(* IEC 61131-3 sources: AXOpen/src/components.abb.robotics/app/src/IO/PLC_LINE, 7 files *)

(* ---- HwIdentifiers.st ---- *)
TYPE
    HwIdentifiers : WORD
    (
        OmniCore_HwID :=	WORD#259,
        OmniCore_DI_64_bytes_DI_64_bytes_HwID :=	WORD#263,
        OmniCore_DO_64_bytes_DO_64_bytes_HwID :=	WORD#262,
        OmniCore_OmniCore_HwID :=	WORD#261,
        OmniCore_OmniCore_OmniCore_Standard_PROFINET_Device_HwID :=	WORD#264,
        OmniCore_OmniCore_profinet_HwID :=	WORD#257,
        OmniCore_OmniCore_profinet_Network_Port_1_HwID :=	WORD#258,
        OmniCore_Rack_HwID :=	WORD#260,
        PROFINET_IO_System_HwID :=	WORD#256,
        RobotBasicIO_HwID :=	WORD#267,
        RobotBasicIO_DI_64_bytes_DI_64_bytes_HwID :=	WORD#271,
        RobotBasicIO_DO_64_bytes_DO_64_bytes_HwID :=	WORD#270,
        RobotBasicIO_Rack_HwID :=	WORD#268,
        RobotBasicIO_RobotBasicIO_HwID :=	WORD#269,
        RobotBasicIO_RobotBasicIO_Robot_Basic_Device_HwID :=	WORD#272,
        RobotBasicIO_RobotBasicIO_profinet_HwID :=	WORD#265,
        RobotBasicIO_RobotBasicIO_profinet_Network_Port_HwID :=	WORD#266,
        plc_line_HwID :=	WORD#32,
        plc_line_Rail_0_HwID :=	WORD#273,
        plc_line_plc_line_HwID :=	WORD#48,
        plc_line_plc_line_CPU_display_1_HwID :=	WORD#54,
        plc_line_plc_line_Card_reader_writer_1_HwID :=	WORD#51,
        plc_line_plc_line_DP_interface_1_HwID :=	WORD#60,
        plc_line_plc_line_OPC_UA_1_HwID :=	WORD#117,
        plc_line_plc_line_PROFINET_interface_X1_HwID :=	WORD#64,
        plc_line_plc_line_PROFINET_interface_X1_Port_1_HwID :=	WORD#65,
        plc_line_plc_line_PROFINET_interface_X1_Port_2_HwID :=	WORD#66,
        plc_line_plc_line_PROFINET_interface_X2_HwID :=	WORD#72,
        plc_line_plc_line_PROFINET_interface_X2_Port_3_HwID :=	WORD#73,
        plc_line_plc_line_Virtual_communication_interface_HwID :=	WORD#135,
        plc_line_plc_line_plc_line_HwID :=	WORD#50,

        NONE := WORD#0
    );
END_TYPE

(* ---- HwInputs.st ---- *)
TYPE
	HwInputs : STRUCT
		RobotBasicIO_DI_64_bytes_1 AT %B0 : ARRAY[0..63] OF BYTE;
		OmniCore_DI_64_bytes_1 AT %B64 : ARRAY[0..63] OF BYTE;
	END_STRUCT;
END_TYPE

(* ---- HwOutputs.st ---- *)
TYPE
	HwOutputs : STRUCT
		RobotBasicIO_DO_64_bytes_1 AT %B0 : ARRAY[0..63] OF BYTE;
		OmniCore_DO_64_bytes_1 AT %B64 : ARRAY[0..63] OF BYTE;
	END_STRUCT;
END_TYPE

(* ---- PlcInputs.st ---- *)
TYPE
	PlcInputs : STRUCT
		RobotBasicIO_DI_64_bytes_1 : ARRAY[0..63] OF BYTE;
		OmniCore_DI_64_bytes_1 : ARRAY[0..63] OF BYTE;
	END_STRUCT;
END_TYPE

(* ---- PlcOutputs.st ---- *)
TYPE
	PlcOutputs : STRUCT
		RobotBasicIO_DO_64_bytes_1 : ARRAY[0..63] OF BYTE;
		OmniCore_DO_64_bytes_1 : ARRAY[0..63] OF BYTE;
	END_STRUCT;
END_TYPE

(* ---- CopyInputs.st ---- *)
FUNCTION CopyInputs
	VAR_EXTERNAL
		HwInputs : HwInputs;
		PlcInputs : PlcInputs;
	END_VAR
	PlcInputs.RobotBasicIO_DI_64_bytes_1[0] := HwInputs.RobotBasicIO_DI_64_bytes_1[0];
	PlcInputs.RobotBasicIO_DI_64_bytes_1[1] := HwInputs.RobotBasicIO_DI_64_bytes_1[1];
	PlcInputs.RobotBasicIO_DI_64_bytes_1[2] := HwInputs.RobotBasicIO_DI_64_bytes_1[2];
	PlcInputs.RobotBasicIO_DI_64_bytes_1[3] := HwInputs.RobotBasicIO_DI_64_bytes_1[3];
	PlcInputs.RobotBasicIO_DI_64_bytes_1[4] := HwInputs.RobotBasicIO_DI_64_bytes_1[4];
	PlcInputs.RobotBasicIO_DI_64_bytes_1[5] := HwInputs.RobotBasicIO_DI_64_bytes_1[5];
	PlcInputs.RobotBasicIO_DI_64_bytes_1[6] := HwInputs.RobotBasicIO_DI_64_bytes_1[6];
	PlcInputs.RobotBasicIO_DI_64_bytes_1[7] := HwInputs.RobotBasicIO_DI_64_bytes_1[7];
	PlcInputs.RobotBasicIO_DI_64_bytes_1[8] := HwInputs.RobotBasicIO_DI_64_bytes_1[8];
	PlcInputs.RobotBasicIO_DI_64_bytes_1[9] := HwInputs.RobotBasicIO_DI_64_bytes_1[9];
	PlcInputs.RobotBasicIO_DI_64_bytes_1[10] := HwInputs.RobotBasicIO_DI_64_bytes_1[10];
	PlcInputs.RobotBasicIO_DI_64_bytes_1[11] := HwInputs.RobotBasicIO_DI_64_bytes_1[11];
	PlcInputs.RobotBasicIO_DI_64_bytes_1[12] := HwInputs.RobotBasicIO_DI_64_bytes_1[12];
	PlcInputs.RobotBasicIO_DI_64_bytes_1[13] := HwInputs.RobotBasicIO_DI_64_bytes_1[13];
	PlcInputs.RobotBasicIO_DI_64_bytes_1[14] := HwInputs.RobotBasicIO_DI_64_bytes_1[14];
	PlcInputs.RobotBasicIO_DI_64_bytes_1[15] := HwInputs.RobotBasicIO_DI_64_bytes_1[15];
	PlcInputs.RobotBasicIO_DI_64_bytes_1[16] := HwInputs.RobotBasicIO_DI_64_bytes_1[16];
	PlcInputs.RobotBasicIO_DI_64_bytes_1[17] := HwInputs.RobotBasicIO_DI_64_bytes_1[17];
	PlcInputs.RobotBasicIO_DI_64_bytes_1[18] := HwInputs.RobotBasicIO_DI_64_bytes_1[18];
	PlcInputs.RobotBasicIO_DI_64_bytes_1[19] := HwInputs.RobotBasicIO_DI_64_bytes_1[19];
	PlcInputs.RobotBasicIO_DI_64_bytes_1[20] := HwInputs.RobotBasicIO_DI_64_bytes_1[20];
	PlcInputs.RobotBasicIO_DI_64_bytes_1[21] := HwInputs.RobotBasicIO_DI_64_bytes_1[21];
	PlcInputs.RobotBasicIO_DI_64_bytes_1[22] := HwInputs.RobotBasicIO_DI_64_bytes_1[22];
	PlcInputs.RobotBasicIO_DI_64_bytes_1[23] := HwInputs.RobotBasicIO_DI_64_bytes_1[23];
	PlcInputs.RobotBasicIO_DI_64_bytes_1[24] := HwInputs.RobotBasicIO_DI_64_bytes_1[24];
	PlcInputs.RobotBasicIO_DI_64_bytes_1[25] := HwInputs.RobotBasicIO_DI_64_bytes_1[25];
	PlcInputs.RobotBasicIO_DI_64_bytes_1[26] := HwInputs.RobotBasicIO_DI_64_bytes_1[26];
	PlcInputs.RobotBasicIO_DI_64_bytes_1[27] := HwInputs.RobotBasicIO_DI_64_bytes_1[27];
	PlcInputs.RobotBasicIO_DI_64_bytes_1[28] := HwInputs.RobotBasicIO_DI_64_bytes_1[28];
	PlcInputs.RobotBasicIO_DI_64_bytes_1[29] := HwInputs.RobotBasicIO_DI_64_bytes_1[29];
	PlcInputs.RobotBasicIO_DI_64_bytes_1[30] := HwInputs.RobotBasicIO_DI_64_bytes_1[30];
	PlcInputs.RobotBasicIO_DI_64_bytes_1[31] := HwInputs.RobotBasicIO_DI_64_bytes_1[31];
	PlcInputs.RobotBasicIO_DI_64_bytes_1[32] := HwInputs.RobotBasicIO_DI_64_bytes_1[32];
	PlcInputs.RobotBasicIO_DI_64_bytes_1[33] := HwInputs.RobotBasicIO_DI_64_bytes_1[33];
	PlcInputs.RobotBasicIO_DI_64_bytes_1[34] := HwInputs.RobotBasicIO_DI_64_bytes_1[34];
	PlcInputs.RobotBasicIO_DI_64_bytes_1[35] := HwInputs.RobotBasicIO_DI_64_bytes_1[35];
	PlcInputs.RobotBasicIO_DI_64_bytes_1[36] := HwInputs.RobotBasicIO_DI_64_bytes_1[36];
	PlcInputs.RobotBasicIO_DI_64_bytes_1[37] := HwInputs.RobotBasicIO_DI_64_bytes_1[37];
	PlcInputs.RobotBasicIO_DI_64_bytes_1[38] := HwInputs.RobotBasicIO_DI_64_bytes_1[38];
	PlcInputs.RobotBasicIO_DI_64_bytes_1[39] := HwInputs.RobotBasicIO_DI_64_bytes_1[39];
	PlcInputs.RobotBasicIO_DI_64_bytes_1[40] := HwInputs.RobotBasicIO_DI_64_bytes_1[40];
	PlcInputs.RobotBasicIO_DI_64_bytes_1[41] := HwInputs.RobotBasicIO_DI_64_bytes_1[41];
	PlcInputs.RobotBasicIO_DI_64_bytes_1[42] := HwInputs.RobotBasicIO_DI_64_bytes_1[42];
	PlcInputs.RobotBasicIO_DI_64_bytes_1[43] := HwInputs.RobotBasicIO_DI_64_bytes_1[43];
	PlcInputs.RobotBasicIO_DI_64_bytes_1[44] := HwInputs.RobotBasicIO_DI_64_bytes_1[44];
	PlcInputs.RobotBasicIO_DI_64_bytes_1[45] := HwInputs.RobotBasicIO_DI_64_bytes_1[45];
	PlcInputs.RobotBasicIO_DI_64_bytes_1[46] := HwInputs.RobotBasicIO_DI_64_bytes_1[46];
	PlcInputs.RobotBasicIO_DI_64_bytes_1[47] := HwInputs.RobotBasicIO_DI_64_bytes_1[47];
	PlcInputs.RobotBasicIO_DI_64_bytes_1[48] := HwInputs.RobotBasicIO_DI_64_bytes_1[48];
	PlcInputs.RobotBasicIO_DI_64_bytes_1[49] := HwInputs.RobotBasicIO_DI_64_bytes_1[49];
	PlcInputs.RobotBasicIO_DI_64_bytes_1[50] := HwInputs.RobotBasicIO_DI_64_bytes_1[50];
	PlcInputs.RobotBasicIO_DI_64_bytes_1[51] := HwInputs.RobotBasicIO_DI_64_bytes_1[51];
	PlcInputs.RobotBasicIO_DI_64_bytes_1[52] := HwInputs.RobotBasicIO_DI_64_bytes_1[52];
	PlcInputs.RobotBasicIO_DI_64_bytes_1[53] := HwInputs.RobotBasicIO_DI_64_bytes_1[53];
	PlcInputs.RobotBasicIO_DI_64_bytes_1[54] := HwInputs.RobotBasicIO_DI_64_bytes_1[54];
	PlcInputs.RobotBasicIO_DI_64_bytes_1[55] := HwInputs.RobotBasicIO_DI_64_bytes_1[55];
	PlcInputs.RobotBasicIO_DI_64_bytes_1[56] := HwInputs.RobotBasicIO_DI_64_bytes_1[56];
	PlcInputs.RobotBasicIO_DI_64_bytes_1[57] := HwInputs.RobotBasicIO_DI_64_bytes_1[57];
	PlcInputs.RobotBasicIO_DI_64_bytes_1[58] := HwInputs.RobotBasicIO_DI_64_bytes_1[58];
	PlcInputs.RobotBasicIO_DI_64_bytes_1[59] := HwInputs.RobotBasicIO_DI_64_bytes_1[59];
	PlcInputs.RobotBasicIO_DI_64_bytes_1[60] := HwInputs.RobotBasicIO_DI_64_bytes_1[60];
	PlcInputs.RobotBasicIO_DI_64_bytes_1[61] := HwInputs.RobotBasicIO_DI_64_bytes_1[61];
	PlcInputs.RobotBasicIO_DI_64_bytes_1[62] := HwInputs.RobotBasicIO_DI_64_bytes_1[62];
	PlcInputs.RobotBasicIO_DI_64_bytes_1[63] := HwInputs.RobotBasicIO_DI_64_bytes_1[63];
	PlcInputs.OmniCore_DI_64_bytes_1[0] := HwInputs.OmniCore_DI_64_bytes_1[0];
	PlcInputs.OmniCore_DI_64_bytes_1[1] := HwInputs.OmniCore_DI_64_bytes_1[1];
	PlcInputs.OmniCore_DI_64_bytes_1[2] := HwInputs.OmniCore_DI_64_bytes_1[2];
	PlcInputs.OmniCore_DI_64_bytes_1[3] := HwInputs.OmniCore_DI_64_bytes_1[3];
	PlcInputs.OmniCore_DI_64_bytes_1[4] := HwInputs.OmniCore_DI_64_bytes_1[4];
	PlcInputs.OmniCore_DI_64_bytes_1[5] := HwInputs.OmniCore_DI_64_bytes_1[5];
	PlcInputs.OmniCore_DI_64_bytes_1[6] := HwInputs.OmniCore_DI_64_bytes_1[6];
	PlcInputs.OmniCore_DI_64_bytes_1[7] := HwInputs.OmniCore_DI_64_bytes_1[7];
	PlcInputs.OmniCore_DI_64_bytes_1[8] := HwInputs.OmniCore_DI_64_bytes_1[8];
	PlcInputs.OmniCore_DI_64_bytes_1[9] := HwInputs.OmniCore_DI_64_bytes_1[9];
	PlcInputs.OmniCore_DI_64_bytes_1[10] := HwInputs.OmniCore_DI_64_bytes_1[10];
	PlcInputs.OmniCore_DI_64_bytes_1[11] := HwInputs.OmniCore_DI_64_bytes_1[11];
	PlcInputs.OmniCore_DI_64_bytes_1[12] := HwInputs.OmniCore_DI_64_bytes_1[12];
	PlcInputs.OmniCore_DI_64_bytes_1[13] := HwInputs.OmniCore_DI_64_bytes_1[13];
	PlcInputs.OmniCore_DI_64_bytes_1[14] := HwInputs.OmniCore_DI_64_bytes_1[14];
	PlcInputs.OmniCore_DI_64_bytes_1[15] := HwInputs.OmniCore_DI_64_bytes_1[15];
	PlcInputs.OmniCore_DI_64_bytes_1[16] := HwInputs.OmniCore_DI_64_bytes_1[16];
	PlcInputs.OmniCore_DI_64_bytes_1[17] := HwInputs.OmniCore_DI_64_bytes_1[17];
	PlcInputs.OmniCore_DI_64_bytes_1[18] := HwInputs.OmniCore_DI_64_bytes_1[18];
	PlcInputs.OmniCore_DI_64_bytes_1[19] := HwInputs.OmniCore_DI_64_bytes_1[19];
	PlcInputs.OmniCore_DI_64_bytes_1[20] := HwInputs.OmniCore_DI_64_bytes_1[20];
	PlcInputs.OmniCore_DI_64_bytes_1[21] := HwInputs.OmniCore_DI_64_bytes_1[21];
	PlcInputs.OmniCore_DI_64_bytes_1[22] := HwInputs.OmniCore_DI_64_bytes_1[22];
	PlcInputs.OmniCore_DI_64_bytes_1[23] := HwInputs.OmniCore_DI_64_bytes_1[23];
	PlcInputs.OmniCore_DI_64_bytes_1[24] := HwInputs.OmniCore_DI_64_bytes_1[24];
	PlcInputs.OmniCore_DI_64_bytes_1[25] := HwInputs.OmniCore_DI_64_bytes_1[25];
	PlcInputs.OmniCore_DI_64_bytes_1[26] := HwInputs.OmniCore_DI_64_bytes_1[26];
	PlcInputs.OmniCore_DI_64_bytes_1[27] := HwInputs.OmniCore_DI_64_bytes_1[27];
	PlcInputs.OmniCore_DI_64_bytes_1[28] := HwInputs.OmniCore_DI_64_bytes_1[28];
	PlcInputs.OmniCore_DI_64_bytes_1[29] := HwInputs.OmniCore_DI_64_bytes_1[29];
	PlcInputs.OmniCore_DI_64_bytes_1[30] := HwInputs.OmniCore_DI_64_bytes_1[30];
	PlcInputs.OmniCore_DI_64_bytes_1[31] := HwInputs.OmniCore_DI_64_bytes_1[31];
	PlcInputs.OmniCore_DI_64_bytes_1[32] := HwInputs.OmniCore_DI_64_bytes_1[32];
	PlcInputs.OmniCore_DI_64_bytes_1[33] := HwInputs.OmniCore_DI_64_bytes_1[33];
	PlcInputs.OmniCore_DI_64_bytes_1[34] := HwInputs.OmniCore_DI_64_bytes_1[34];
	PlcInputs.OmniCore_DI_64_bytes_1[35] := HwInputs.OmniCore_DI_64_bytes_1[35];
	PlcInputs.OmniCore_DI_64_bytes_1[36] := HwInputs.OmniCore_DI_64_bytes_1[36];
	PlcInputs.OmniCore_DI_64_bytes_1[37] := HwInputs.OmniCore_DI_64_bytes_1[37];
	PlcInputs.OmniCore_DI_64_bytes_1[38] := HwInputs.OmniCore_DI_64_bytes_1[38];
	PlcInputs.OmniCore_DI_64_bytes_1[39] := HwInputs.OmniCore_DI_64_bytes_1[39];
	PlcInputs.OmniCore_DI_64_bytes_1[40] := HwInputs.OmniCore_DI_64_bytes_1[40];
	PlcInputs.OmniCore_DI_64_bytes_1[41] := HwInputs.OmniCore_DI_64_bytes_1[41];
	PlcInputs.OmniCore_DI_64_bytes_1[42] := HwInputs.OmniCore_DI_64_bytes_1[42];
	PlcInputs.OmniCore_DI_64_bytes_1[43] := HwInputs.OmniCore_DI_64_bytes_1[43];
	PlcInputs.OmniCore_DI_64_bytes_1[44] := HwInputs.OmniCore_DI_64_bytes_1[44];
	PlcInputs.OmniCore_DI_64_bytes_1[45] := HwInputs.OmniCore_DI_64_bytes_1[45];
	PlcInputs.OmniCore_DI_64_bytes_1[46] := HwInputs.OmniCore_DI_64_bytes_1[46];
	PlcInputs.OmniCore_DI_64_bytes_1[47] := HwInputs.OmniCore_DI_64_bytes_1[47];
	PlcInputs.OmniCore_DI_64_bytes_1[48] := HwInputs.OmniCore_DI_64_bytes_1[48];
	PlcInputs.OmniCore_DI_64_bytes_1[49] := HwInputs.OmniCore_DI_64_bytes_1[49];
	PlcInputs.OmniCore_DI_64_bytes_1[50] := HwInputs.OmniCore_DI_64_bytes_1[50];
	PlcInputs.OmniCore_DI_64_bytes_1[51] := HwInputs.OmniCore_DI_64_bytes_1[51];
	PlcInputs.OmniCore_DI_64_bytes_1[52] := HwInputs.OmniCore_DI_64_bytes_1[52];
	PlcInputs.OmniCore_DI_64_bytes_1[53] := HwInputs.OmniCore_DI_64_bytes_1[53];
	PlcInputs.OmniCore_DI_64_bytes_1[54] := HwInputs.OmniCore_DI_64_bytes_1[54];
	PlcInputs.OmniCore_DI_64_bytes_1[55] := HwInputs.OmniCore_DI_64_bytes_1[55];
	PlcInputs.OmniCore_DI_64_bytes_1[56] := HwInputs.OmniCore_DI_64_bytes_1[56];
	PlcInputs.OmniCore_DI_64_bytes_1[57] := HwInputs.OmniCore_DI_64_bytes_1[57];
	PlcInputs.OmniCore_DI_64_bytes_1[58] := HwInputs.OmniCore_DI_64_bytes_1[58];
	PlcInputs.OmniCore_DI_64_bytes_1[59] := HwInputs.OmniCore_DI_64_bytes_1[59];
	PlcInputs.OmniCore_DI_64_bytes_1[60] := HwInputs.OmniCore_DI_64_bytes_1[60];
	PlcInputs.OmniCore_DI_64_bytes_1[61] := HwInputs.OmniCore_DI_64_bytes_1[61];
	PlcInputs.OmniCore_DI_64_bytes_1[62] := HwInputs.OmniCore_DI_64_bytes_1[62];
	PlcInputs.OmniCore_DI_64_bytes_1[63] := HwInputs.OmniCore_DI_64_bytes_1[63];
END_FUNCTION

(* ---- CopyOutputs.st ---- *)
FUNCTION CopyOutputs
	VAR_EXTERNAL
		HwOutputs : HwOutputs;
		PlcOutputs : PlcOutputs;
	END_VAR
	HwOutputs.RobotBasicIO_DO_64_bytes_1[0] := PlcOutputs.RobotBasicIO_DO_64_bytes_1[0];
	HwOutputs.RobotBasicIO_DO_64_bytes_1[1] := PlcOutputs.RobotBasicIO_DO_64_bytes_1[1];
	HwOutputs.RobotBasicIO_DO_64_bytes_1[2] := PlcOutputs.RobotBasicIO_DO_64_bytes_1[2];
	HwOutputs.RobotBasicIO_DO_64_bytes_1[3] := PlcOutputs.RobotBasicIO_DO_64_bytes_1[3];
	HwOutputs.RobotBasicIO_DO_64_bytes_1[4] := PlcOutputs.RobotBasicIO_DO_64_bytes_1[4];
	HwOutputs.RobotBasicIO_DO_64_bytes_1[5] := PlcOutputs.RobotBasicIO_DO_64_bytes_1[5];
	HwOutputs.RobotBasicIO_DO_64_bytes_1[6] := PlcOutputs.RobotBasicIO_DO_64_bytes_1[6];
	HwOutputs.RobotBasicIO_DO_64_bytes_1[7] := PlcOutputs.RobotBasicIO_DO_64_bytes_1[7];
	HwOutputs.RobotBasicIO_DO_64_bytes_1[8] := PlcOutputs.RobotBasicIO_DO_64_bytes_1[8];
	HwOutputs.RobotBasicIO_DO_64_bytes_1[9] := PlcOutputs.RobotBasicIO_DO_64_bytes_1[9];
	HwOutputs.RobotBasicIO_DO_64_bytes_1[10] := PlcOutputs.RobotBasicIO_DO_64_bytes_1[10];
	HwOutputs.RobotBasicIO_DO_64_bytes_1[11] := PlcOutputs.RobotBasicIO_DO_64_bytes_1[11];
	HwOutputs.RobotBasicIO_DO_64_bytes_1[12] := PlcOutputs.RobotBasicIO_DO_64_bytes_1[12];
	HwOutputs.RobotBasicIO_DO_64_bytes_1[13] := PlcOutputs.RobotBasicIO_DO_64_bytes_1[13];
	HwOutputs.RobotBasicIO_DO_64_bytes_1[14] := PlcOutputs.RobotBasicIO_DO_64_bytes_1[14];
	HwOutputs.RobotBasicIO_DO_64_bytes_1[15] := PlcOutputs.RobotBasicIO_DO_64_bytes_1[15];
	HwOutputs.RobotBasicIO_DO_64_bytes_1[16] := PlcOutputs.RobotBasicIO_DO_64_bytes_1[16];
	HwOutputs.RobotBasicIO_DO_64_bytes_1[17] := PlcOutputs.RobotBasicIO_DO_64_bytes_1[17];
	HwOutputs.RobotBasicIO_DO_64_bytes_1[18] := PlcOutputs.RobotBasicIO_DO_64_bytes_1[18];
	HwOutputs.RobotBasicIO_DO_64_bytes_1[19] := PlcOutputs.RobotBasicIO_DO_64_bytes_1[19];
	HwOutputs.RobotBasicIO_DO_64_bytes_1[20] := PlcOutputs.RobotBasicIO_DO_64_bytes_1[20];
	HwOutputs.RobotBasicIO_DO_64_bytes_1[21] := PlcOutputs.RobotBasicIO_DO_64_bytes_1[21];
	HwOutputs.RobotBasicIO_DO_64_bytes_1[22] := PlcOutputs.RobotBasicIO_DO_64_bytes_1[22];
	HwOutputs.RobotBasicIO_DO_64_bytes_1[23] := PlcOutputs.RobotBasicIO_DO_64_bytes_1[23];
	HwOutputs.RobotBasicIO_DO_64_bytes_1[24] := PlcOutputs.RobotBasicIO_DO_64_bytes_1[24];
	HwOutputs.RobotBasicIO_DO_64_bytes_1[25] := PlcOutputs.RobotBasicIO_DO_64_bytes_1[25];
	HwOutputs.RobotBasicIO_DO_64_bytes_1[26] := PlcOutputs.RobotBasicIO_DO_64_bytes_1[26];
	HwOutputs.RobotBasicIO_DO_64_bytes_1[27] := PlcOutputs.RobotBasicIO_DO_64_bytes_1[27];
	HwOutputs.RobotBasicIO_DO_64_bytes_1[28] := PlcOutputs.RobotBasicIO_DO_64_bytes_1[28];
	HwOutputs.RobotBasicIO_DO_64_bytes_1[29] := PlcOutputs.RobotBasicIO_DO_64_bytes_1[29];
	HwOutputs.RobotBasicIO_DO_64_bytes_1[30] := PlcOutputs.RobotBasicIO_DO_64_bytes_1[30];
	HwOutputs.RobotBasicIO_DO_64_bytes_1[31] := PlcOutputs.RobotBasicIO_DO_64_bytes_1[31];
	HwOutputs.RobotBasicIO_DO_64_bytes_1[32] := PlcOutputs.RobotBasicIO_DO_64_bytes_1[32];
	HwOutputs.RobotBasicIO_DO_64_bytes_1[33] := PlcOutputs.RobotBasicIO_DO_64_bytes_1[33];
	HwOutputs.RobotBasicIO_DO_64_bytes_1[34] := PlcOutputs.RobotBasicIO_DO_64_bytes_1[34];
	HwOutputs.RobotBasicIO_DO_64_bytes_1[35] := PlcOutputs.RobotBasicIO_DO_64_bytes_1[35];
	HwOutputs.RobotBasicIO_DO_64_bytes_1[36] := PlcOutputs.RobotBasicIO_DO_64_bytes_1[36];
	HwOutputs.RobotBasicIO_DO_64_bytes_1[37] := PlcOutputs.RobotBasicIO_DO_64_bytes_1[37];
	HwOutputs.RobotBasicIO_DO_64_bytes_1[38] := PlcOutputs.RobotBasicIO_DO_64_bytes_1[38];
	HwOutputs.RobotBasicIO_DO_64_bytes_1[39] := PlcOutputs.RobotBasicIO_DO_64_bytes_1[39];
	HwOutputs.RobotBasicIO_DO_64_bytes_1[40] := PlcOutputs.RobotBasicIO_DO_64_bytes_1[40];
	HwOutputs.RobotBasicIO_DO_64_bytes_1[41] := PlcOutputs.RobotBasicIO_DO_64_bytes_1[41];
	HwOutputs.RobotBasicIO_DO_64_bytes_1[42] := PlcOutputs.RobotBasicIO_DO_64_bytes_1[42];
	HwOutputs.RobotBasicIO_DO_64_bytes_1[43] := PlcOutputs.RobotBasicIO_DO_64_bytes_1[43];
	HwOutputs.RobotBasicIO_DO_64_bytes_1[44] := PlcOutputs.RobotBasicIO_DO_64_bytes_1[44];
	HwOutputs.RobotBasicIO_DO_64_bytes_1[45] := PlcOutputs.RobotBasicIO_DO_64_bytes_1[45];
	HwOutputs.RobotBasicIO_DO_64_bytes_1[46] := PlcOutputs.RobotBasicIO_DO_64_bytes_1[46];
	HwOutputs.RobotBasicIO_DO_64_bytes_1[47] := PlcOutputs.RobotBasicIO_DO_64_bytes_1[47];
	HwOutputs.RobotBasicIO_DO_64_bytes_1[48] := PlcOutputs.RobotBasicIO_DO_64_bytes_1[48];
	HwOutputs.RobotBasicIO_DO_64_bytes_1[49] := PlcOutputs.RobotBasicIO_DO_64_bytes_1[49];
	HwOutputs.RobotBasicIO_DO_64_bytes_1[50] := PlcOutputs.RobotBasicIO_DO_64_bytes_1[50];
	HwOutputs.RobotBasicIO_DO_64_bytes_1[51] := PlcOutputs.RobotBasicIO_DO_64_bytes_1[51];
	HwOutputs.RobotBasicIO_DO_64_bytes_1[52] := PlcOutputs.RobotBasicIO_DO_64_bytes_1[52];
	HwOutputs.RobotBasicIO_DO_64_bytes_1[53] := PlcOutputs.RobotBasicIO_DO_64_bytes_1[53];
	HwOutputs.RobotBasicIO_DO_64_bytes_1[54] := PlcOutputs.RobotBasicIO_DO_64_bytes_1[54];
	HwOutputs.RobotBasicIO_DO_64_bytes_1[55] := PlcOutputs.RobotBasicIO_DO_64_bytes_1[55];
	HwOutputs.RobotBasicIO_DO_64_bytes_1[56] := PlcOutputs.RobotBasicIO_DO_64_bytes_1[56];
	HwOutputs.RobotBasicIO_DO_64_bytes_1[57] := PlcOutputs.RobotBasicIO_DO_64_bytes_1[57];
	HwOutputs.RobotBasicIO_DO_64_bytes_1[58] := PlcOutputs.RobotBasicIO_DO_64_bytes_1[58];
	HwOutputs.RobotBasicIO_DO_64_bytes_1[59] := PlcOutputs.RobotBasicIO_DO_64_bytes_1[59];
	HwOutputs.RobotBasicIO_DO_64_bytes_1[60] := PlcOutputs.RobotBasicIO_DO_64_bytes_1[60];
	HwOutputs.RobotBasicIO_DO_64_bytes_1[61] := PlcOutputs.RobotBasicIO_DO_64_bytes_1[61];
	HwOutputs.RobotBasicIO_DO_64_bytes_1[62] := PlcOutputs.RobotBasicIO_DO_64_bytes_1[62];
	HwOutputs.RobotBasicIO_DO_64_bytes_1[63] := PlcOutputs.RobotBasicIO_DO_64_bytes_1[63];
	HwOutputs.OmniCore_DO_64_bytes_1[0] := PlcOutputs.OmniCore_DO_64_bytes_1[0];
	HwOutputs.OmniCore_DO_64_bytes_1[1] := PlcOutputs.OmniCore_DO_64_bytes_1[1];
	HwOutputs.OmniCore_DO_64_bytes_1[2] := PlcOutputs.OmniCore_DO_64_bytes_1[2];
	HwOutputs.OmniCore_DO_64_bytes_1[3] := PlcOutputs.OmniCore_DO_64_bytes_1[3];
	HwOutputs.OmniCore_DO_64_bytes_1[4] := PlcOutputs.OmniCore_DO_64_bytes_1[4];
	HwOutputs.OmniCore_DO_64_bytes_1[5] := PlcOutputs.OmniCore_DO_64_bytes_1[5];
	HwOutputs.OmniCore_DO_64_bytes_1[6] := PlcOutputs.OmniCore_DO_64_bytes_1[6];
	HwOutputs.OmniCore_DO_64_bytes_1[7] := PlcOutputs.OmniCore_DO_64_bytes_1[7];
	HwOutputs.OmniCore_DO_64_bytes_1[8] := PlcOutputs.OmniCore_DO_64_bytes_1[8];
	HwOutputs.OmniCore_DO_64_bytes_1[9] := PlcOutputs.OmniCore_DO_64_bytes_1[9];
	HwOutputs.OmniCore_DO_64_bytes_1[10] := PlcOutputs.OmniCore_DO_64_bytes_1[10];
	HwOutputs.OmniCore_DO_64_bytes_1[11] := PlcOutputs.OmniCore_DO_64_bytes_1[11];
	HwOutputs.OmniCore_DO_64_bytes_1[12] := PlcOutputs.OmniCore_DO_64_bytes_1[12];
	HwOutputs.OmniCore_DO_64_bytes_1[13] := PlcOutputs.OmniCore_DO_64_bytes_1[13];
	HwOutputs.OmniCore_DO_64_bytes_1[14] := PlcOutputs.OmniCore_DO_64_bytes_1[14];
	HwOutputs.OmniCore_DO_64_bytes_1[15] := PlcOutputs.OmniCore_DO_64_bytes_1[15];
	HwOutputs.OmniCore_DO_64_bytes_1[16] := PlcOutputs.OmniCore_DO_64_bytes_1[16];
	HwOutputs.OmniCore_DO_64_bytes_1[17] := PlcOutputs.OmniCore_DO_64_bytes_1[17];
	HwOutputs.OmniCore_DO_64_bytes_1[18] := PlcOutputs.OmniCore_DO_64_bytes_1[18];
	HwOutputs.OmniCore_DO_64_bytes_1[19] := PlcOutputs.OmniCore_DO_64_bytes_1[19];
	HwOutputs.OmniCore_DO_64_bytes_1[20] := PlcOutputs.OmniCore_DO_64_bytes_1[20];
	HwOutputs.OmniCore_DO_64_bytes_1[21] := PlcOutputs.OmniCore_DO_64_bytes_1[21];
	HwOutputs.OmniCore_DO_64_bytes_1[22] := PlcOutputs.OmniCore_DO_64_bytes_1[22];
	HwOutputs.OmniCore_DO_64_bytes_1[23] := PlcOutputs.OmniCore_DO_64_bytes_1[23];
	HwOutputs.OmniCore_DO_64_bytes_1[24] := PlcOutputs.OmniCore_DO_64_bytes_1[24];
	HwOutputs.OmniCore_DO_64_bytes_1[25] := PlcOutputs.OmniCore_DO_64_bytes_1[25];
	HwOutputs.OmniCore_DO_64_bytes_1[26] := PlcOutputs.OmniCore_DO_64_bytes_1[26];
	HwOutputs.OmniCore_DO_64_bytes_1[27] := PlcOutputs.OmniCore_DO_64_bytes_1[27];
	HwOutputs.OmniCore_DO_64_bytes_1[28] := PlcOutputs.OmniCore_DO_64_bytes_1[28];
	HwOutputs.OmniCore_DO_64_bytes_1[29] := PlcOutputs.OmniCore_DO_64_bytes_1[29];
	HwOutputs.OmniCore_DO_64_bytes_1[30] := PlcOutputs.OmniCore_DO_64_bytes_1[30];
	HwOutputs.OmniCore_DO_64_bytes_1[31] := PlcOutputs.OmniCore_DO_64_bytes_1[31];
	HwOutputs.OmniCore_DO_64_bytes_1[32] := PlcOutputs.OmniCore_DO_64_bytes_1[32];
	HwOutputs.OmniCore_DO_64_bytes_1[33] := PlcOutputs.OmniCore_DO_64_bytes_1[33];
	HwOutputs.OmniCore_DO_64_bytes_1[34] := PlcOutputs.OmniCore_DO_64_bytes_1[34];
	HwOutputs.OmniCore_DO_64_bytes_1[35] := PlcOutputs.OmniCore_DO_64_bytes_1[35];
	HwOutputs.OmniCore_DO_64_bytes_1[36] := PlcOutputs.OmniCore_DO_64_bytes_1[36];
	HwOutputs.OmniCore_DO_64_bytes_1[37] := PlcOutputs.OmniCore_DO_64_bytes_1[37];
	HwOutputs.OmniCore_DO_64_bytes_1[38] := PlcOutputs.OmniCore_DO_64_bytes_1[38];
	HwOutputs.OmniCore_DO_64_bytes_1[39] := PlcOutputs.OmniCore_DO_64_bytes_1[39];
	HwOutputs.OmniCore_DO_64_bytes_1[40] := PlcOutputs.OmniCore_DO_64_bytes_1[40];
	HwOutputs.OmniCore_DO_64_bytes_1[41] := PlcOutputs.OmniCore_DO_64_bytes_1[41];
	HwOutputs.OmniCore_DO_64_bytes_1[42] := PlcOutputs.OmniCore_DO_64_bytes_1[42];
	HwOutputs.OmniCore_DO_64_bytes_1[43] := PlcOutputs.OmniCore_DO_64_bytes_1[43];
	HwOutputs.OmniCore_DO_64_bytes_1[44] := PlcOutputs.OmniCore_DO_64_bytes_1[44];
	HwOutputs.OmniCore_DO_64_bytes_1[45] := PlcOutputs.OmniCore_DO_64_bytes_1[45];
	HwOutputs.OmniCore_DO_64_bytes_1[46] := PlcOutputs.OmniCore_DO_64_bytes_1[46];
	HwOutputs.OmniCore_DO_64_bytes_1[47] := PlcOutputs.OmniCore_DO_64_bytes_1[47];
	HwOutputs.OmniCore_DO_64_bytes_1[48] := PlcOutputs.OmniCore_DO_64_bytes_1[48];
	HwOutputs.OmniCore_DO_64_bytes_1[49] := PlcOutputs.OmniCore_DO_64_bytes_1[49];
	HwOutputs.OmniCore_DO_64_bytes_1[50] := PlcOutputs.OmniCore_DO_64_bytes_1[50];
	HwOutputs.OmniCore_DO_64_bytes_1[51] := PlcOutputs.OmniCore_DO_64_bytes_1[51];
	HwOutputs.OmniCore_DO_64_bytes_1[52] := PlcOutputs.OmniCore_DO_64_bytes_1[52];
	HwOutputs.OmniCore_DO_64_bytes_1[53] := PlcOutputs.OmniCore_DO_64_bytes_1[53];
	HwOutputs.OmniCore_DO_64_bytes_1[54] := PlcOutputs.OmniCore_DO_64_bytes_1[54];
	HwOutputs.OmniCore_DO_64_bytes_1[55] := PlcOutputs.OmniCore_DO_64_bytes_1[55];
	HwOutputs.OmniCore_DO_64_bytes_1[56] := PlcOutputs.OmniCore_DO_64_bytes_1[56];
	HwOutputs.OmniCore_DO_64_bytes_1[57] := PlcOutputs.OmniCore_DO_64_bytes_1[57];
	HwOutputs.OmniCore_DO_64_bytes_1[58] := PlcOutputs.OmniCore_DO_64_bytes_1[58];
	HwOutputs.OmniCore_DO_64_bytes_1[59] := PlcOutputs.OmniCore_DO_64_bytes_1[59];
	HwOutputs.OmniCore_DO_64_bytes_1[60] := PlcOutputs.OmniCore_DO_64_bytes_1[60];
	HwOutputs.OmniCore_DO_64_bytes_1[61] := PlcOutputs.OmniCore_DO_64_bytes_1[61];
	HwOutputs.OmniCore_DO_64_bytes_1[62] := PlcOutputs.OmniCore_DO_64_bytes_1[62];
	HwOutputs.OmniCore_DO_64_bytes_1[63] := PlcOutputs.OmniCore_DO_64_bytes_1[63];
END_FUNCTION
